Staubli VAL3: getEvent.pgx

public program getEvent(string& x_sItem, num x_nIndex, num x_nBoxType)
  local num i
  local string l_sKey
begin

  switch x_nBoxType
    case 1
      // start from the first
      l_sKey=first(sml:box)
      // search it
      while l_sKey!=""
        x_sItem=l_sKey
        l_sKey=next(sml:box[l_sKey])
        if i==x_nIndex
          return
        else
          i=i+1
        endIf
      endWhile
    break
    case 2
      // start from the first
      l_sKey=first(big:box)
      // search it
      while l_sKey!=""
        x_sItem=l_sKey
        l_sKey=next(big:box[l_sKey])
        if i==x_nIndex
          return
        else
          i=i+1
        endIf
      endWhile
    break
  endSwitch
end
